(* IEC 61131-3 sources: CodesysTest/export/UN00 - Sharp Bagger/EM02 - Discharge/IEM02_Discharge.itf, 1 file *)

(* ---- TakeAwayBag.m.st ---- *)
(*#-#-#-#-#-#-#-#-#-#---Declaration---#-#-#-#-#-#-#-#-#-#-#-#-#*)

METHOD TakeAwayBag
VAR_INPUT
	caller : IAllObjects;
END_VAR
